Fanuc KAREL source: kt00402.compact.KL

PROGRAM KT00402
%STACKSIZE=65535
%PRIORITY=65535
%NOLOCKGROUP
VAR
I1 : INTEGER
R2 : REAL
OUT : BOOLEAN
BEGIN
I1=2
R2=3.0
OUT=((I1) > R2)
END KT00402
